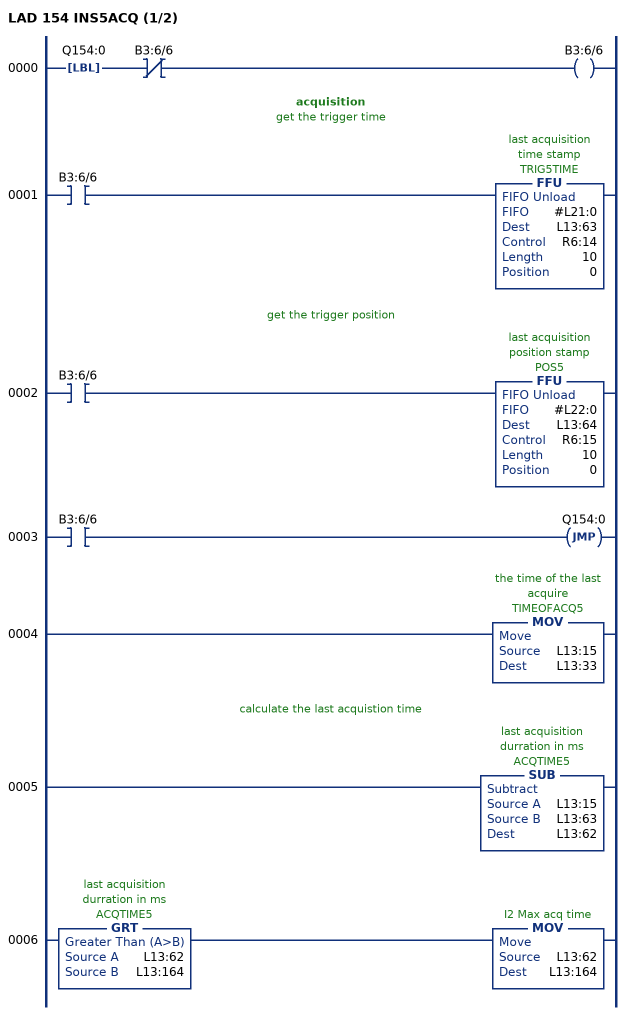
% Rung: 0 %
SOR LBL Q154:0 XIO B3:6/6 OTE B3:6/6 EOR
% Rung: 1 %
% TITLE: acquisition %
% get the trigger time %
SOR XIC B3:6/6 FFU #L21:0 L13:63 R6:14 10 0 EOR
%   L13:63  TRIG5TIME  "last acquisition time stamp" %
% Rung: 2 %
% get the trigger position %
SOR XIC B3:6/6 FFU #L22:0 L13:64 R6:15 10 0 EOR
%   L13:64  POS5  "last acquisition position stamp" %
% Rung: 3 %
SOR XIC B3:6/6 JMP Q154:0 EOR
% Rung: 4 %
SOR MOV L13:15 L13:33 EOR
%   L13:15  THE_TIME %
%   L13:33  TIMEOFACQ5  "the time of the last acquire" %
% Rung: 5 %
% calculate the last acquistion time %
SOR SUB L13:15 L13:63 L13:62 EOR
%   L13:15  THE_TIME %
%   L13:63  TRIG5TIME  "last acquisition time stamp" %
%   L13:62  ACQTIME5  "last acquisition durration in ms" %
% Rung: 6 %
SOR GRT L13:62 L13:164 MOV L13:62 L13:164 EOR
%   L13:62  ACQTIME5  "last acquisition durration in ms" %
%   L13:164  "I2 Max acq time" %

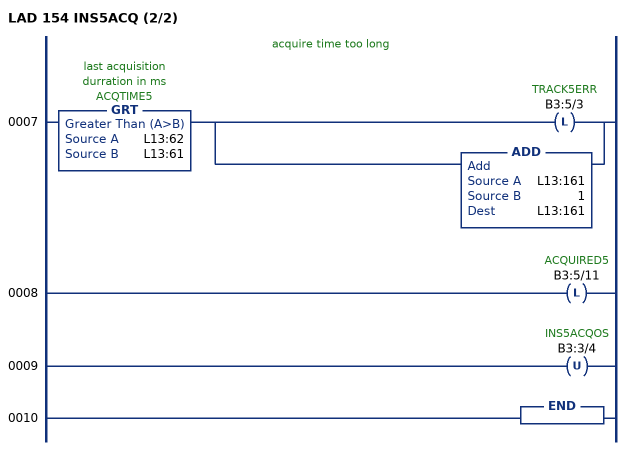
% Rung: 7 %
% acquire time too long %
SOR GRT L13:62 L13:61 BST OTL B3:5/3 NXB ADD L13:161 1 L13:161 BND EOR
%   L13:62  ACQTIME5  "last acquisition durration in ms" %
%   L13:61  "max acquisition time in ms" %
%   B3:5/3  TRACK5ERR %
% Rung: 8 %
SOR OTL B3:5/11 EOR
%   B3:5/11  ACQUIRED5 %
% Rung: 9 %
SOR OTU B3:3/4 EOR
%   B3:3/4  INS5ACQOS %
% Rung: 10 %
SOR END EOR

LADDER 155 "INS5TRIG"
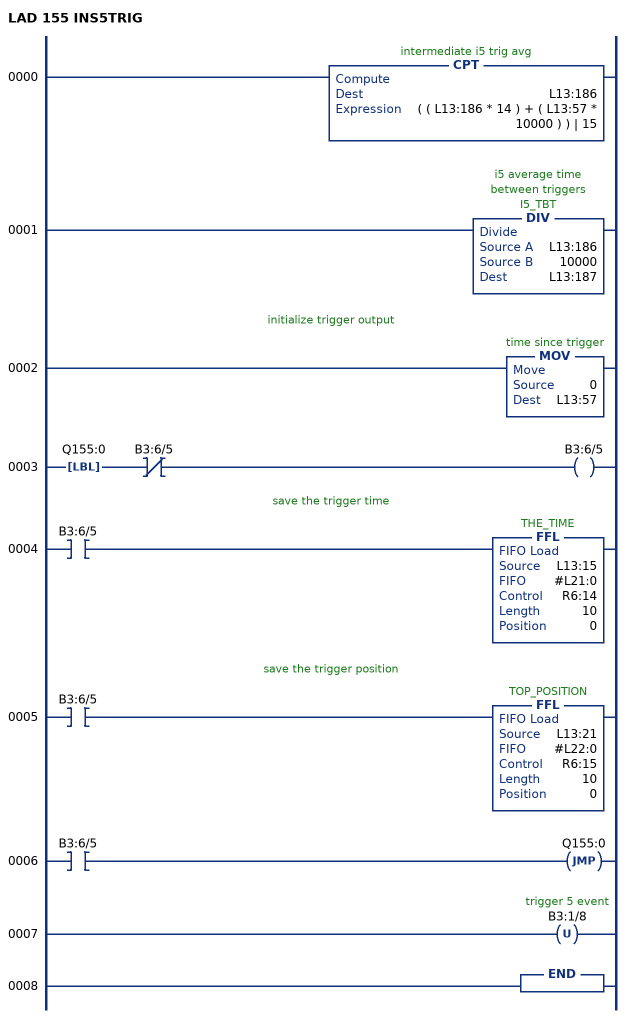
% Rung: 0 %
SOR CPT L13:186 " ( ( L13:186 * 14 ) + ( L13:57 * 10000 ) ) | 15 " EOR
%   L13:186  "intermediate i5 trig avg" %
%   L13:57  "time since trigger" %
% Rung: 1 %
SOR DIV L13:186 10000 L13:187 EOR
%   L13:186  "intermediate i5 trig avg" %
%   L13:187  I5_TBT  "i5 average time between triggers" %
% Rung: 2 %
% initialize trigger output %
SOR MOV 0 L13:57 EOR
%   L13:57  "time since trigger" %
% Rung: 3 %
SOR LBL Q155:0 XIO B3:6/5 OTE B3:6/5 EOR
% Rung: 4 %
% save the trigger time %
SOR XIC B3:6/5 FFL L13:15 #L21:0 R6:14 10 0 EOR
%   L13:15  THE_TIME %
% Rung: 5 %
% save the trigger position %
SOR XIC B3:6/5 FFL L13:21 #L22:0 R6:15 10 0 EOR
%   L13:21  TOP_POSITION %
% Rung: 6 %
SOR XIC B3:6/5 JMP Q155:0 EOR
% Rung: 7 %
SOR OTU B3:1/8 EOR
%   B3:1/8  "trigger 5 event" %
% Rung: 8 %
SOR END EOR

LADDER 159 "INS6RESULT"
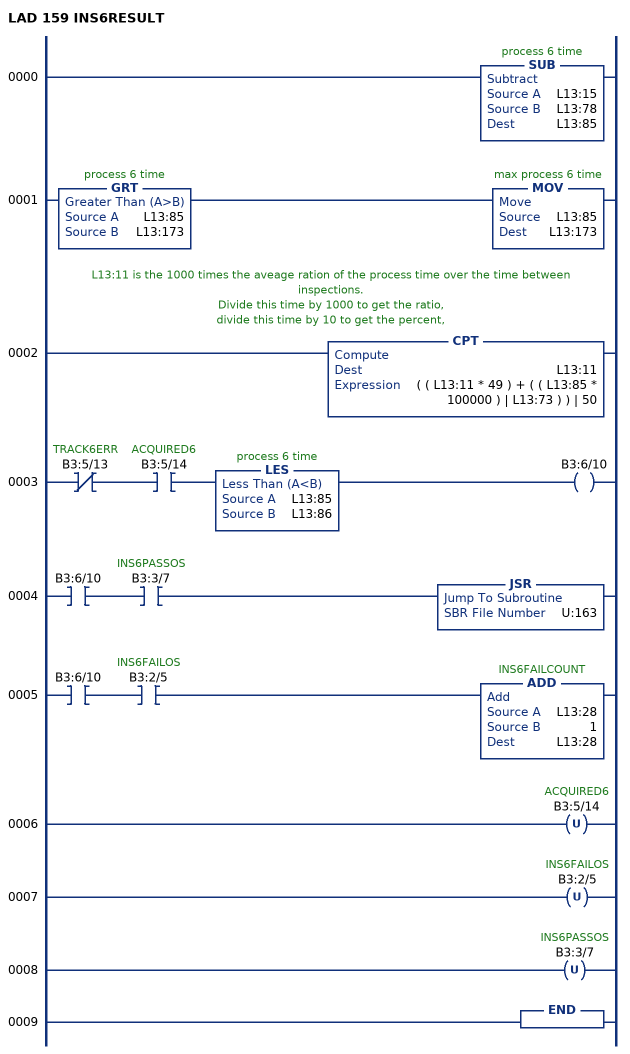
% Rung: 0 %
SOR SUB L13:15 L13:78 L13:85 EOR
%   L13:15  THE_TIME %
%   L13:78  TIMEOFACQ6  "the time of the last acquire" %
%   L13:85  "process 6 time" %
% Rung: 1 %
SOR GRT L13:85 L13:173 MOV L13:85 L13:173 EOR
%   L13:85  "process 6 time" %
%   L13:173  "max process 6 time" %
% Rung: 2 %
% L13:11 is the 1000 times the aveage ration of the process time over the time between inspections.
% Divide this time by 1000 to get the ratio,
% divide this time by 10 to get the percent, %
SOR CPT L13:11 " ( ( L13:11 * 49 ) + ( ( L13:85 * 100000 ) | L13:73 ) ) | 50 " EOR
%   L13:85  "process 6 time" %
%   L13:73  TBI  "the time between inspections in 0.000,01 seconds or 1/6000000 minutes." %
% Rung: 3 %
SOR XIO B3:5/13 XIC B3:5/14 LES L13:85 L13:86 OTE B3:6/10 EOR
%   B3:5/13  TRACK6ERR %
%   B3:5/14  ACQUIRED6 %
%   L13:85  "process 6 time" %
% Rung: 4 %
SOR XIC B3:6/10 XIC B3:3/7 JSR U:163 EOR
%   B3:3/7  INS6PASSOS %
% Rung: 5 %
SOR XIC B3:6/10 XIC B3:2/5 ADD L13:28 1 L13:28 EOR
%   B3:2/5  INS6FAILOS %
%   L13:28  INS6FAILCOUNT %
% Rung: 6 %
SOR OTU B3:5/14 EOR
%   B3:5/14  ACQUIRED6 %
% Rung: 7 %
SOR OTU B3:2/5 EOR
%   B3:2/5  INS6FAILOS %
% Rung: 8 %
SOR OTU B3:3/7 EOR
%   B3:3/7  INS6PASSOS %
% Rung: 9 %
SOR END EOR

LADDER 160 "FIXERR6"
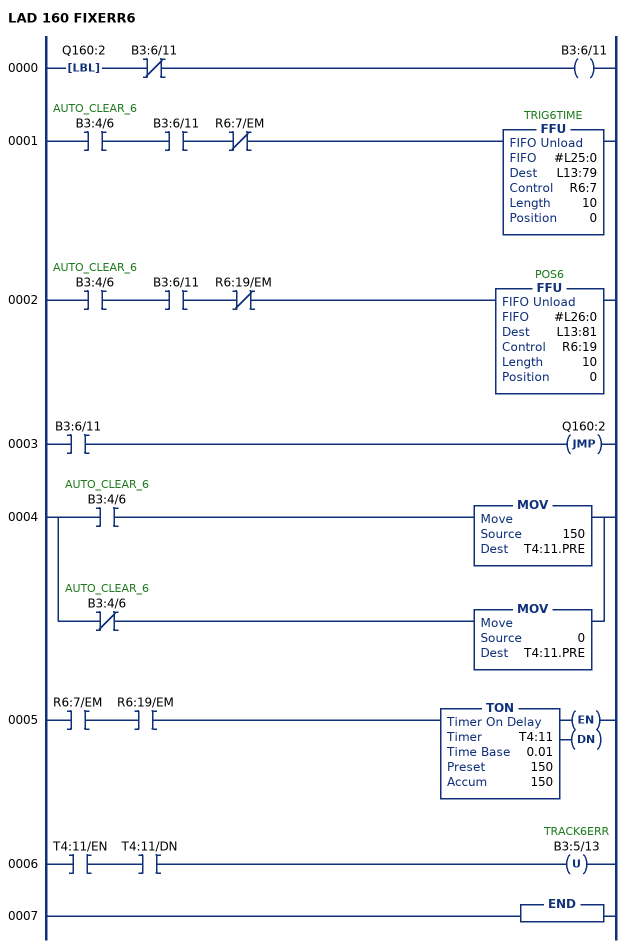
% Rung: 0 %
SOR LBL Q160:2 XIO B3:6/11 OTE B3:6/11 EOR
% Rung: 1 %
SOR XIC B3:4/6 XIC B3:6/11 XIO R6:7/EM FFU #L25:0 L13:79 R6:7 10 0 EOR
%   B3:4/6  AUTO_CLEAR_6 %
%   L13:79  TRIG6TIME %
% Rung: 2 %
SOR XIC B3:4/6 XIC B3:6/11 XIO R6:19/EM FFU #L26:0 L13:81 R6:19 10 0 EOR
%   B3:4/6  AUTO_CLEAR_6 %
%   L13:81  POS6 %
% Rung: 3 %
SOR XIC B3:6/11 JMP Q160:2 EOR
% Rung: 4 %
SOR BST XIC B3:4/6 MOV 150 T4:11.PRE NXB XIO B3:4/6 MOV 0 T4:11.PRE BND EOR
%   B3:4/6  AUTO_CLEAR_6 %
% Rung: 5 %
SOR XIC R6:7/EM XIC R6:19/EM TON T4:11 0.01 150 150 EOR
% Rung: 6 %
SOR XIC T4:11/EN XIC T4:11/DN OTU B3:5/13 EOR
%   B3:5/13  TRACK6ERR %
% Rung: 7 %
SOR END EOR

LADDER 162 "INS6"
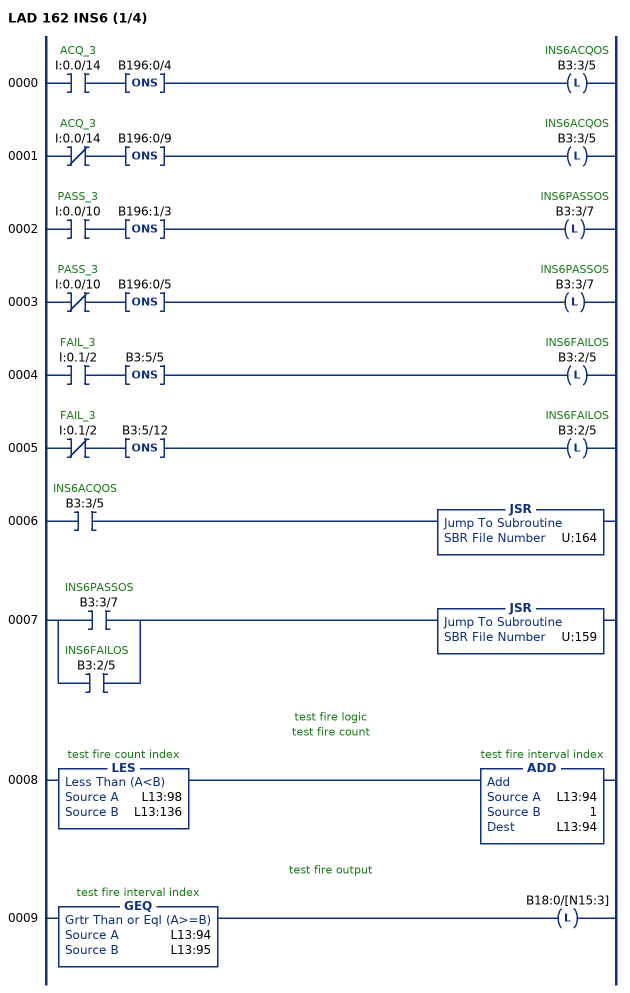
% Rung: 0 %
SOR XIC I:0.0/14 ONS B196:0/4 OTL B3:3/5 EOR
%   I:0.0/14  ACQ_3 %
%   B3:3/5  INS6ACQOS %
% Rung: 1 %
SOR XIO I:0.0/14 ONS B196:0/9 OTL B3:3/5 EOR
%   I:0.0/14  ACQ_3 %
%   B3:3/5  INS6ACQOS %
% Rung: 2 %
SOR XIC I:0.0/10 ONS B196:1/3 OTL B3:3/7 EOR
%   I:0.0/10  PASS_3 %
%   B3:3/7  INS6PASSOS %
% Rung: 3 %
SOR XIO I:0.0/10 ONS B196:0/5 OTL B3:3/7 EOR
%   I:0.0/10  PASS_3 %
%   B3:3/7  INS6PASSOS %
% Rung: 4 %
SOR XIC I:0.1/2 ONS B3:5/5 OTL B3:2/5 EOR
%   I:0.1/2  FAIL_3 %
%   B3:2/5  INS6FAILOS %
% Rung: 5 %
SOR XIO I:0.1/2 ONS B3:5/12 OTL B3:2/5 EOR
%   I:0.1/2  FAIL_3 %
%   B3:2/5  INS6FAILOS %
% Rung: 6 %
SOR XIC B3:3/5 JSR U:164 EOR
%   B3:3/5  INS6ACQOS %
% Rung: 7 %
SOR BST XIC B3:3/7 NXB XIC B3:2/5 BND JSR U:159 EOR
%   B3:3/7  INS6PASSOS %
%   B3:2/5  INS6FAILOS %
% Rung: 8 %
% test fire logic
% 
% test fire count %
SOR LES L13:98 L13:136 ADD L13:94 1 L13:94 EOR
%   L13:98  "test fire count index" %
%   L13:136  "test fire count" %
%   L13:94  "test fire interval index" %
% Rung: 9 %
% test fire output %
SOR GEQ L13:94 L13:95 OTL B18:0/[N15:3] EOR
%   L13:94  "test fire interval index" %
%   L13:95  "test fire interval" %
%   N15:3  INS_6_TRIG_LOC %

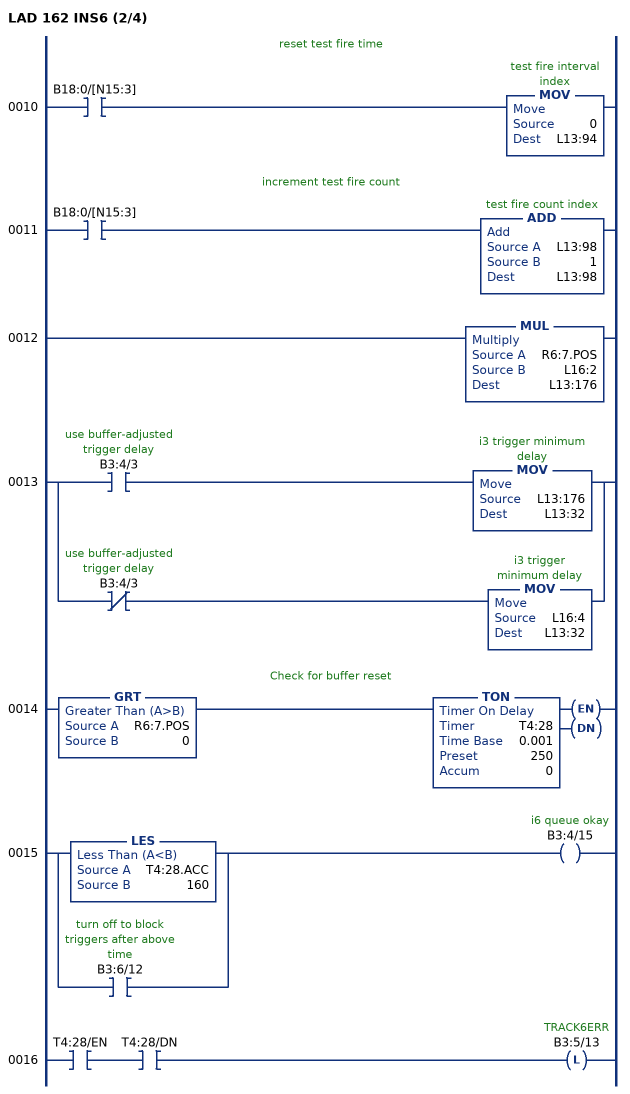
% Rung: 10 %
% reset test fire time %
SOR XIC B18:0/[N15:3] MOV 0 L13:94 EOR
%   N15:3  INS_6_TRIG_LOC %
%   L13:94  "test fire interval index" %
% Rung: 11 %
% increment test fire count %
SOR XIC B18:0/[N15:3] ADD L13:98 1 L13:98 EOR
%   N15:3  INS_6_TRIG_LOC %
%   L13:98  "test fire count index" %
% Rung: 12 %
SOR MUL R6:7.POS L16:2 L13:176 EOR
%   L16:2  TRIG_DELAY_Q_MULTI %
% Rung: 13 %
SOR BST XIC B3:4/3 MOV L13:176 L13:32 NXB XIO B3:4/3 MOV L16:4 L13:32 BND EOR
%   B3:4/3  "use buffer-adjusted trigger delay" %
%   L13:32  "i3 trigger minimum delay" %
%   L16:4  TRIG_DELAY_FLAT_RATE %
% Rung: 14 %
% Check for buffer reset %
SOR GRT R6:7.POS 0 TON T4:28 0.001 250 0 EOR
% Rung: 15 %
SOR BST LES T4:28.ACC 160 NXB XIC B3:6/12 BND OTE B3:4/15 EOR
%   B3:6/12  "turn off to block triggers after above time" %
%   B3:4/15  "i6 queue okay" %
% Rung: 16 %
SOR XIC T4:28/EN XIC T4:28/DN OTL B3:5/13 EOR
%   B3:5/13  TRACK6ERR %

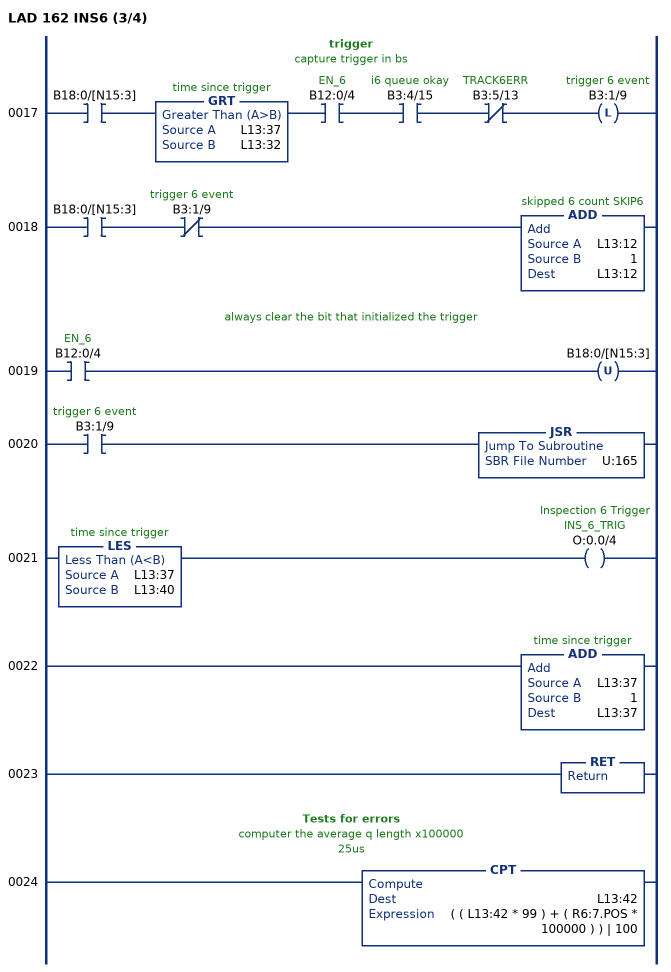
% Rung: 17 %
% TITLE: trigger %
% capture trigger in bs %
SOR XIC B18:0/[N15:3] GRT L13:37 L13:32 XIC B12:0/4 XIC B3:4/15 XIO B3:5/13 OTL B3:1/9 EOR
%   N15:3  INS_6_TRIG_LOC %
%   L13:37  "time since trigger" %
%   L13:32  "i3 trigger minimum delay" %
%   B12:0/4  EN_6 %
%   B3:4/15  "i6 queue okay" %
%   B3:5/13  TRACK6ERR %
%   B3:1/9  "trigger 6 event" %
% Rung: 18 %
SOR XIC B18:0/[N15:3] XIO B3:1/9 ADD L13:12 1 L13:12 EOR
%   N15:3  INS_6_TRIG_LOC %
%   B3:1/9  "trigger 6 event" %
%   L13:12  SKIP6  "skipped 6 count" %
% Rung: 19 %
% always clear the bit that initialized the trigger %
SOR XIC B12:0/4 OTU B18:0/[N15:3] EOR
%   B12:0/4  EN_6 %
%   N15:3  INS_6_TRIG_LOC %
% Rung: 20 %
SOR XIC B3:1/9 JSR U:165 EOR
%   B3:1/9  "trigger 6 event" %
% Rung: 21 %
SOR LES L13:37 L13:40 OTE O:0.0/4 EOR
%   L13:37  "time since trigger" %
%   L13:40  "last part time" %
%   O:0.0/4  INS_6_TRIG  "Inspection 6 Trigger" %
% Rung: 22 %
SOR ADD L13:37 1 L13:37 EOR
%   L13:37  "time since trigger" %
% Rung: 23 %
SOR RET EOR
% Rung: 24 %
% TITLE: Tests for errors %
% computer the average q length x100000
% 25us %
SOR CPT L13:42 " ( ( L13:42 * 99 ) + ( R6:7.POS * 100000 ) ) | 100 " EOR

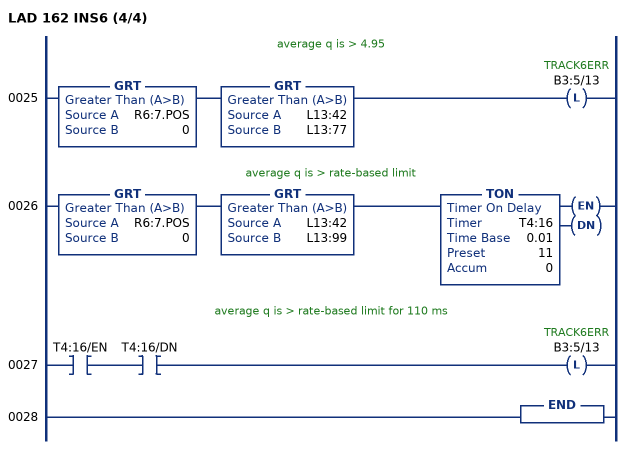
% Rung: 25 %
% average q is > 4.95 %
SOR GRT R6:7.POS 0 GRT L13:42 L13:77 OTL B3:5/13 EOR
%   B3:5/13  TRACK6ERR %
% Rung: 26 %
% average q is > rate-based limit %
SOR GRT R6:7.POS 0 GRT L13:42 L13:99 TON T4:16 0.01 11 0 EOR
%   L13:99  "i6 timed queue limit" %
% Rung: 27 %
% average q is > rate-based limit for 110 ms %
SOR XIC T4:16/EN XIC T4:16/DN OTL B3:5/13 EOR
%   B3:5/13  TRACK6ERR %
% Rung: 28 %
SOR END EOR

LADDER 163 "INS6PASS"
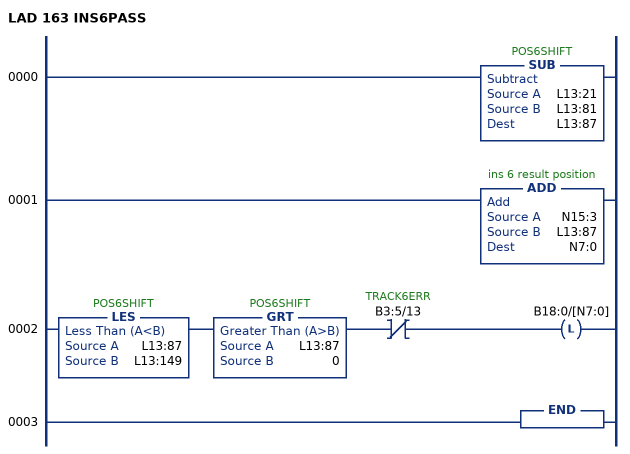
% Rung: 0 %
SOR SUB L13:21 L13:81 L13:87 EOR
%   L13:21  TOP_POSITION %
%   L13:81  POS6 %
%   L13:87  POS6SHIFT %
% Rung: 1 %
SOR ADD N15:3 L13:87 N7:0 EOR
%   N15:3  INS_6_TRIG_LOC %
%   L13:87  POS6SHIFT %
%   N7:0  "ins 6 result position" %
% Rung: 2 %
SOR LES L13:87 L13:149 GRT L13:87 0 XIO B3:5/13 OTL B18:0/[N7:0] EOR
%   L13:87  POS6SHIFT %
%   B3:5/13  TRACK6ERR %
%   N7:0  "ins 6 result position" %
% Rung: 3 %
SOR END EOR

LADDER 164 "INS6ACQ"
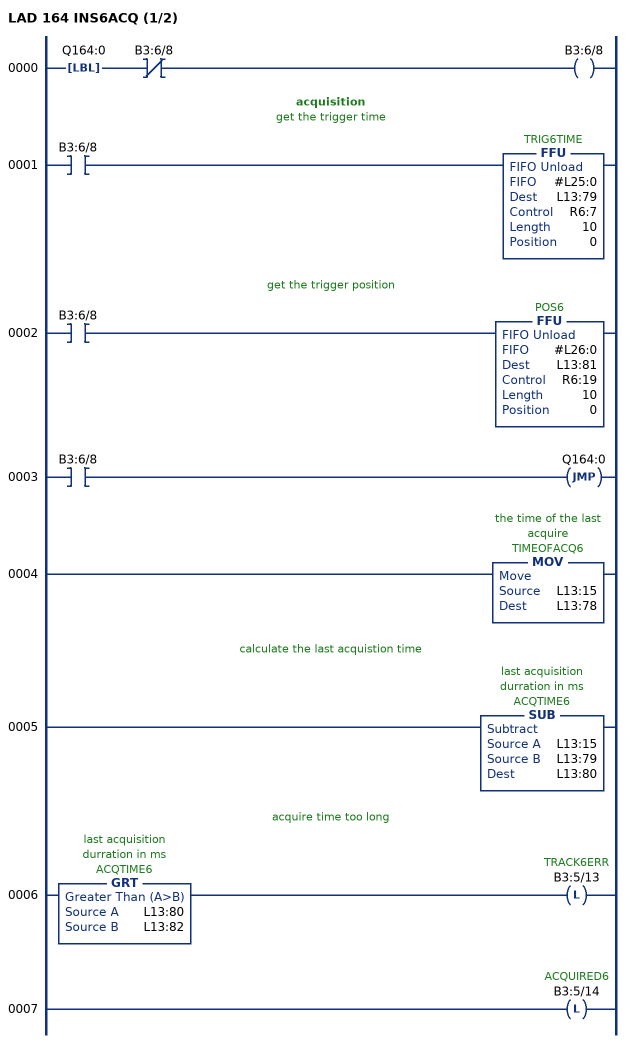
% Rung: 0 %
SOR LBL Q164:0 XIO B3:6/8 OTE B3:6/8 EOR
% Rung: 1 %
% TITLE: acquisition %
% get the trigger time %
SOR XIC B3:6/8 FFU #L25:0 L13:79 R6:7 10 0 EOR
%   L13:79  TRIG6TIME %
% Rung: 2 %
% get the trigger position %
SOR XIC B3:6/8 FFU #L26:0 L13:81 R6:19 10 0 EOR
%   L13:81  POS6 %
% Rung: 3 %
SOR XIC B3:6/8 JMP Q164:0 EOR
% Rung: 4 %
SOR MOV L13:15 L13:78 EOR
%   L13:15  THE_TIME %
%   L13:78  TIMEOFACQ6  "the time of the last acquire" %
% Rung: 5 %
% calculate the last acquistion time %
SOR SUB L13:15 L13:79 L13:80 EOR
%   L13:15  THE_TIME %
%   L13:79  TRIG6TIME %
%   L13:80  ACQTIME6  "last acquisition durration in ms" %
% Rung: 6 %
% acquire time too long %
SOR GRT L13:80 L13:82 OTL B3:5/13 EOR
%   L13:80  ACQTIME6  "last acquisition durration in ms" %
%   B3:5/13  TRACK6ERR %
% Rung: 7 %
SOR OTL B3:5/14 EOR
%   B3:5/14  ACQUIRED6 %

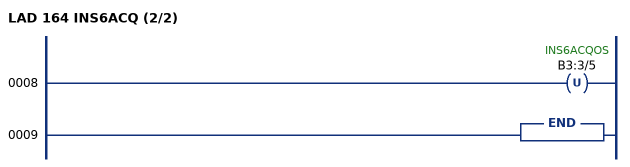
% Rung: 8 %
SOR OTU B3:3/5 EOR
%   B3:3/5  INS6ACQOS %
% Rung: 9 %
SOR END EOR

LADDER 165 "INS6TRIG"
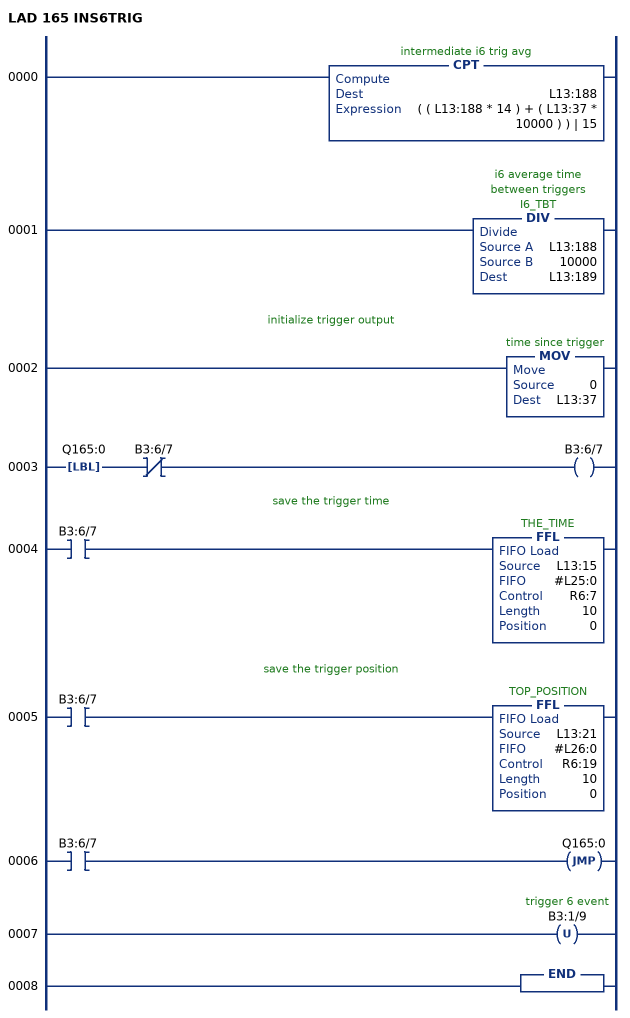
% Rung: 0 %
SOR CPT L13:188 " ( ( L13:188 * 14 ) + ( L13:37 * 10000 ) ) | 15 " EOR
%   L13:188  "intermediate i6 trig avg" %
%   L13:37  "time since trigger" %
% Rung: 1 %
SOR DIV L13:188 10000 L13:189 EOR
%   L13:188  "intermediate i6 trig avg" %
%   L13:189  I6_TBT  "i6 average time between triggers" %
% Rung: 2 %
% initialize trigger output %
SOR MOV 0 L13:37 EOR
%   L13:37  "time since trigger" %
% Rung: 3 %
SOR LBL Q165:0 XIO B3:6/7 OTE B3:6/7 EOR
% Rung: 4 %
% save the trigger time %
SOR XIC B3:6/7 FFL L13:15 #L25:0 R6:7 10 0 EOR
%   L13:15  THE_TIME %
% Rung: 5 %
% save the trigger position %
SOR XIC B3:6/7 FFL L13:21 #L26:0 R6:19 10 0 EOR
%   L13:21  TOP_POSITION %
% Rung: 6 %
SOR XIC B3:6/7 JMP Q165:0 EOR
% Rung: 7 %
SOR OTU B3:1/9 EOR
%   B3:1/9  "trigger 6 event" %
% Rung: 8 %
SOR END EOR

LADDER 170 "PASS BLOW"
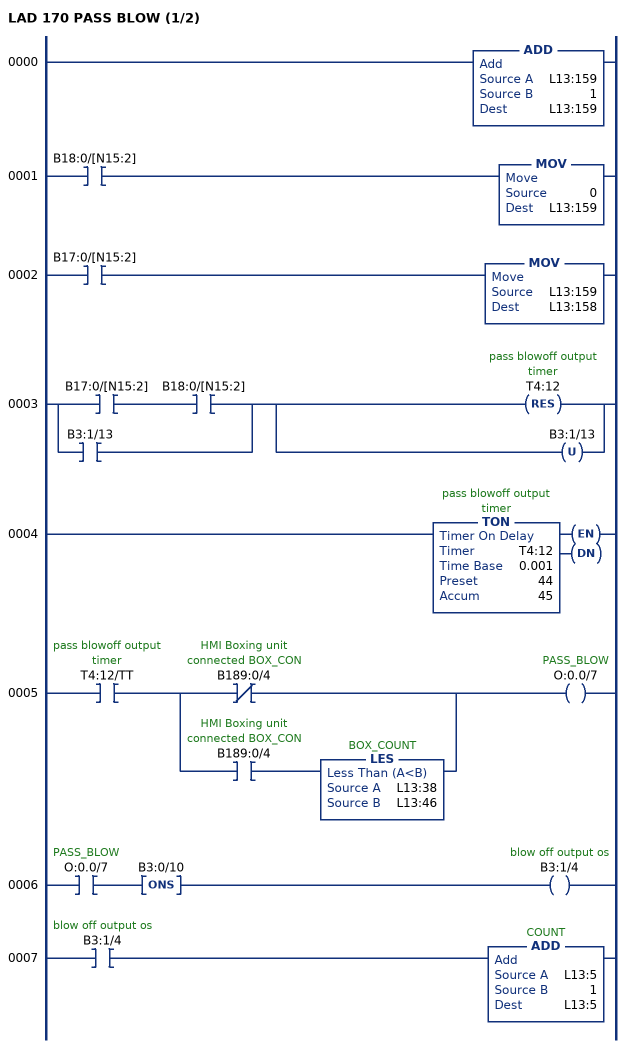
% Rung: 0 %
SOR ADD L13:159 1 L13:159 EOR
% Rung: 1 %
SOR XIC B18:0/[N15:2] MOV 0 L13:159 EOR
%   N15:2  BLOW_PT %
% Rung: 2 %
SOR XIC B17:0/[N15:2] MOV L13:159 L13:158 EOR
%   N15:2  BLOW_PT %
% Rung: 3 %
SOR BST XIC B17:0/[N15:2] XIC B18:0/[N15:2] NXB XIC B3:1/13 BND BST RES T4:12 NXB OTU B3:1/13 BND EOR
%   N15:2  BLOW_PT %
%   T4:12  "pass blowoff output timer" %
% Rung: 4 %
SOR TON T4:12 0.001 44 45 EOR
%   T4:12  "pass blowoff output timer" %
% Rung: 5 %
SOR XIC T4:12/TT BST XIO B189:0/4 NXB XIC B189:0/4 LES L13:38 L13:46 BND OTE O:0.0/7 EOR
%   T4:12  "pass blowoff output timer" %
%   B189:0/4  BOX_CON  "HMI Boxing unit connected" %
%   L13:38  BOX_COUNT %
%   L13:46  BOX_LIMIT  "box count setpoint" %
%   O:0.0/7  PASS_BLOW %
% Rung: 6 %
SOR XIC O:0.0/7 ONS B3:0/10 OTE B3:1/4 EOR
%   O:0.0/7  PASS_BLOW %
%   B3:1/4  "blow off output os" %
% Rung: 7 %
SOR XIC B3:1/4 ADD L13:5 1 L13:5 EOR
%   B3:1/4  "blow off output os" %
%   L13:5  COUNT %

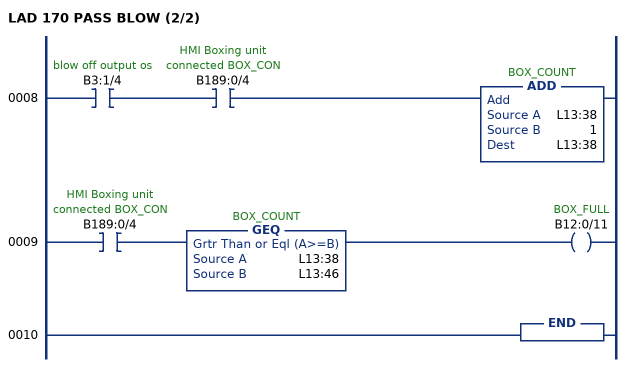
% Rung: 8 %
SOR XIC B3:1/4 XIC B189:0/4 ADD L13:38 1 L13:38 EOR
%   B3:1/4  "blow off output os" %
%   B189:0/4  BOX_CON  "HMI Boxing unit connected" %
%   L13:38  BOX_COUNT %
% Rung: 9 %
SOR XIC B189:0/4 GEQ L13:38 L13:46 OTE B12:0/11 EOR
%   B189:0/4  BOX_CON  "HMI Boxing unit connected" %
%   L13:38  BOX_COUNT %
%   L13:46  BOX_LIMIT  "box count setpoint" %
%   B12:0/11  BOX_FULL %
% Rung: 10 %
SOR END EOR

LADDER 180 "RATE"
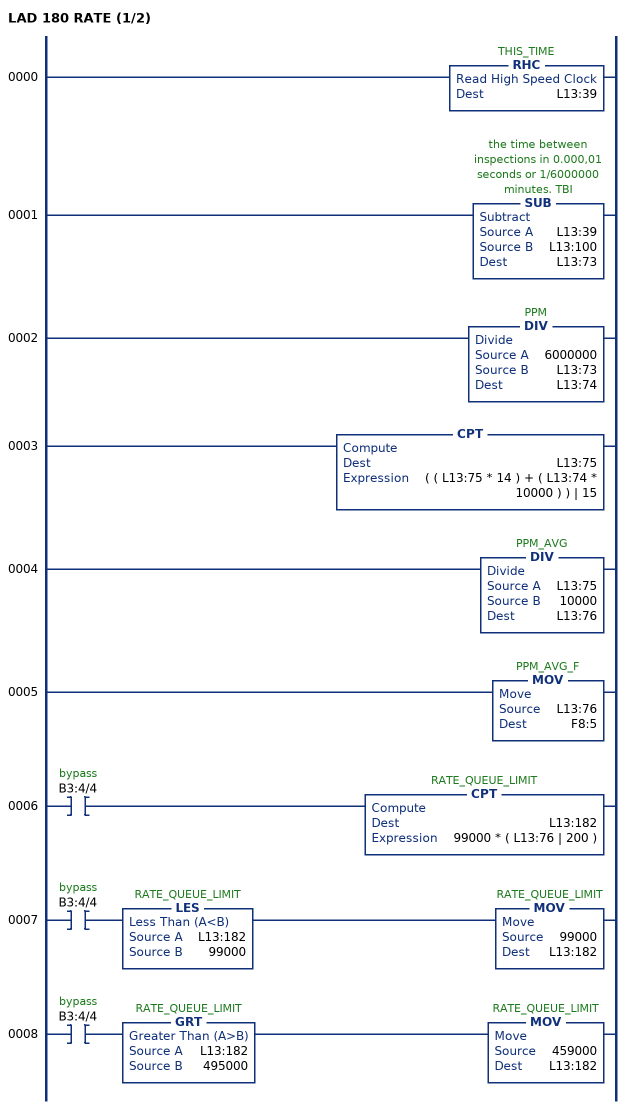
% Rung: 0 %
SOR RHC L13:39 EOR
%   L13:39  THIS_TIME %
% Rung: 1 %
SOR SUB L13:39 L13:100 L13:73 EOR
%   L13:39  THIS_TIME %
%   L13:100  LAST_PART_TIME  "the time clock reading when the previous part was triggered" %
%   L13:73  TBI  "the time between inspections in 0.000,01 seconds or 1/6000000 minutes." %
% Rung: 2 %
SOR DIV 6000000 L13:73 L13:74 EOR
%   L13:73  TBI  "the time between inspections in 0.000,01 seconds or 1/6000000 minutes." %
%   L13:74  PPM %
% Rung: 3 %
SOR CPT L13:75 " ( ( L13:75 * 14 ) + ( L13:74 * 10000 ) ) | 15 " EOR
%   L13:74  PPM %
% Rung: 4 %
SOR DIV L13:75 10000 L13:76 EOR
%   L13:76  PPM_AVG %
% Rung: 5 %
SOR MOV L13:76 F8:5 EOR
%   L13:76  PPM_AVG %
%   F8:5  PPM_AVG_F %
% Rung: 6 %
SOR XIC B3:4/4 CPT L13:182 " 99000 * ( L13:76 | 200 ) " EOR
%   B3:4/4  "bypass" %
%   L13:182  RATE_QUEUE_LIMIT %
%   L13:76  PPM_AVG %
% Rung: 7 %
SOR XIC B3:4/4 LES L13:182 99000 MOV 99000 L13:182 EOR
%   B3:4/4  "bypass" %
%   L13:182  RATE_QUEUE_LIMIT %
% Rung: 8 %
SOR XIC B3:4/4 GRT L13:182 495000 MOV 459000 L13:182 EOR
%   B3:4/4  "bypass" %
%   L13:182  RATE_QUEUE_LIMIT %

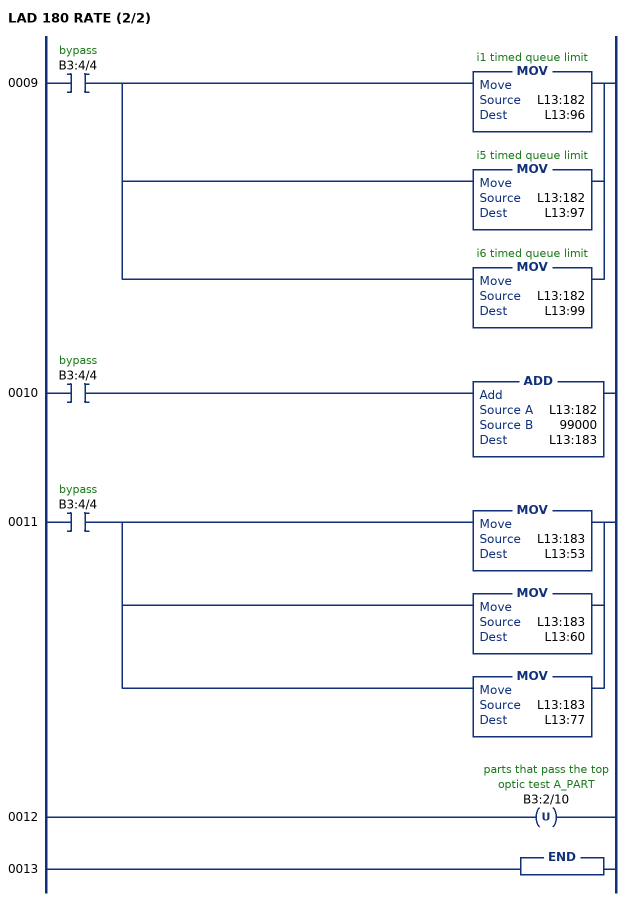
% Rung: 9 %
SOR XIC B3:4/4 BST MOV L13:182 L13:96 NXB MOV L13:182 L13:97 NXB MOV L13:182 L13:99 BND EOR
%   B3:4/4  "bypass" %
%   L13:182  RATE_QUEUE_LIMIT %
%   L13:96  "i1 timed queue limit" %
%   L13:97  "i5 timed queue limit" %
%   L13:99  "i6 timed queue limit" %
% Rung: 10 %
SOR XIC B3:4/4 ADD L13:182 99000 L13:183 EOR
%   B3:4/4  "bypass" %
%   L13:182  RATE_QUEUE_LIMIT %
% Rung: 11 %
SOR XIC B3:4/4 BST MOV L13:183 L13:53 NXB MOV L13:183 L13:60 NXB MOV L13:183 L13:77 BND EOR
%   B3:4/4  "bypass" %
% Rung: 12 %
SOR OTU B3:2/10 EOR
%   B3:2/10  A_PART  "parts that pass the top optic test" %
% Rung: 13 %
SOR END EOR

LADDER 200 "TESTOPTIC"
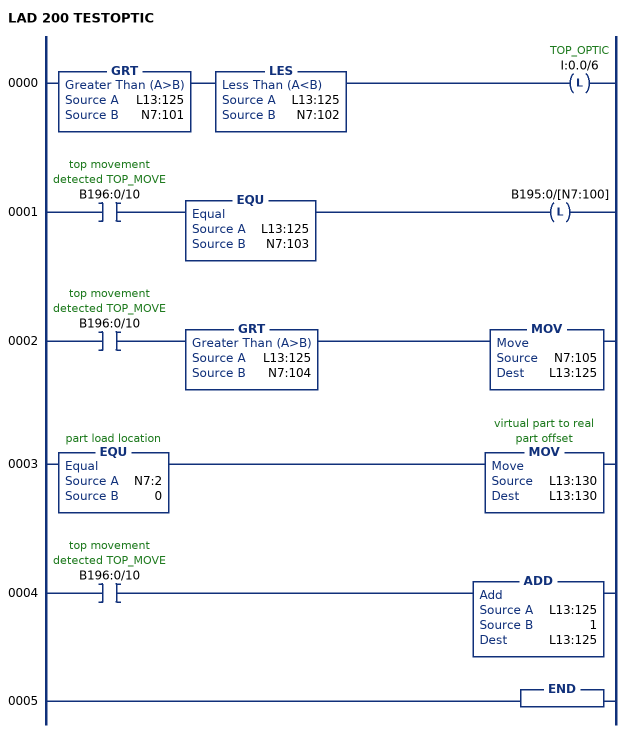
% Rung: 0 %
SOR GRT L13:125 N7:101 LES L13:125 N7:102 OTL I:0.0/6 EOR
%   I:0.0/6  TOP_OPTIC %
% Rung: 1 %
SOR XIC B196:0/10 EQU L13:125 N7:103 OTL B195:0/[N7:100] EOR
%   B196:0/10  TOP_MOVE  "top movement detected" %
% Rung: 2 %
SOR XIC B196:0/10 GRT L13:125 N7:104 MOV N7:105 L13:125 EOR
%   B196:0/10  TOP_MOVE  "top movement detected" %
% Rung: 3 %
SOR EQU N7:2 0 MOV L13:130 L13:130 EOR
%   N7:2  "part load location" %
%   L13:130  "virtual part to real part offset" %
% Rung: 4 %
SOR XIC B196:0/10 ADD L13:125 1 L13:125 EOR
%   B196:0/10  TOP_MOVE  "top movement detected" %
% Rung: 5 %
SOR END EOR

LADDER 201 "UNUSED"
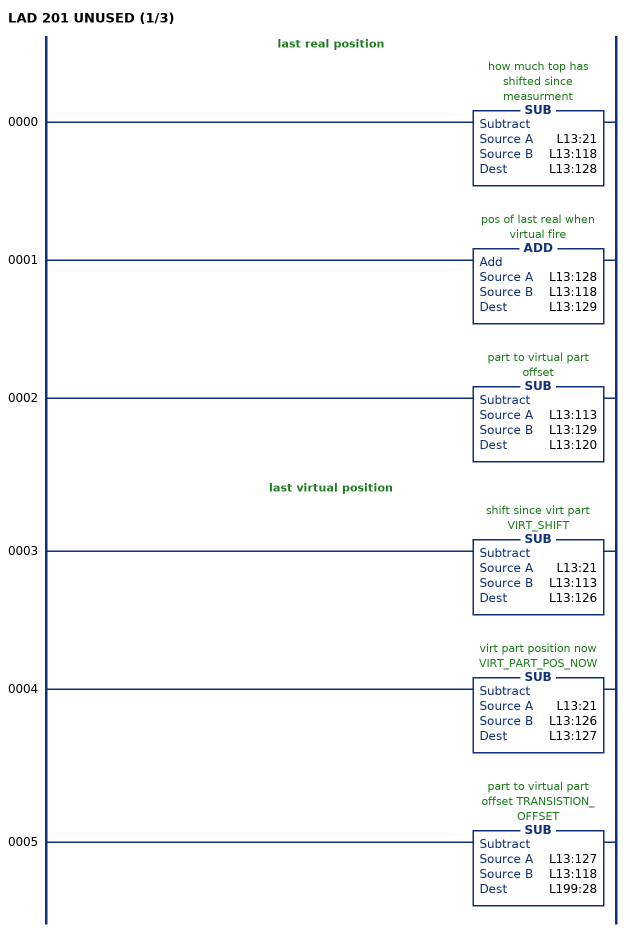
% Rung: 0 %
% TITLE: last real position %
SOR SUB L13:21 L13:118 L13:128 EOR
%   L13:21  TOP_POSITION %
%   L13:118  REAL_PT_RAW_CL  "real part center line in raw position" %
%   L13:128  "how much top has shifted since measurment" %
% Rung: 1 %
SOR ADD L13:128 L13:118 L13:129 EOR
%   L13:128  "how much top has shifted since measurment" %
%   L13:118  REAL_PT_RAW_CL  "real part center line in raw position" %
%   L13:129  "pos of last real when virtual fire" %
% Rung: 2 %
SOR SUB L13:113 L13:129 L13:120 EOR
%   L13:113  VERTUAL_PT_RAW_CL  "virtual part center line transfer from the bottom in raw position" %
%   L13:129  "pos of last real when virtual fire" %
%   L13:120  "part to virtual part offset" %
% Rung: 3 %
% TITLE: last virtual position %
SOR SUB L13:21 L13:113 L13:126 EOR
%   L13:21  TOP_POSITION %
%   L13:113  VERTUAL_PT_RAW_CL  "virtual part center line transfer from the bottom in raw position" %
%   L13:126  VIRT_SHIFT  "shift since virt part" %
% Rung: 4 %
SOR SUB L13:21 L13:126 L13:127 EOR
%   L13:21  TOP_POSITION %
%   L13:126  VIRT_SHIFT  "shift since virt part" %
%   L13:127  VIRT_PART_POS_NOW  "virt part position now" %
% Rung: 5 %
SOR SUB L13:127 L13:118 L199:28 EOR
%   L13:127  VIRT_PART_POS_NOW  "virt part position now" %
%   L13:118  REAL_PT_RAW_CL  "real part center line in raw position" %
%   L199:28  TRANSISTION_OFFSET  "part to virtual part offset" %

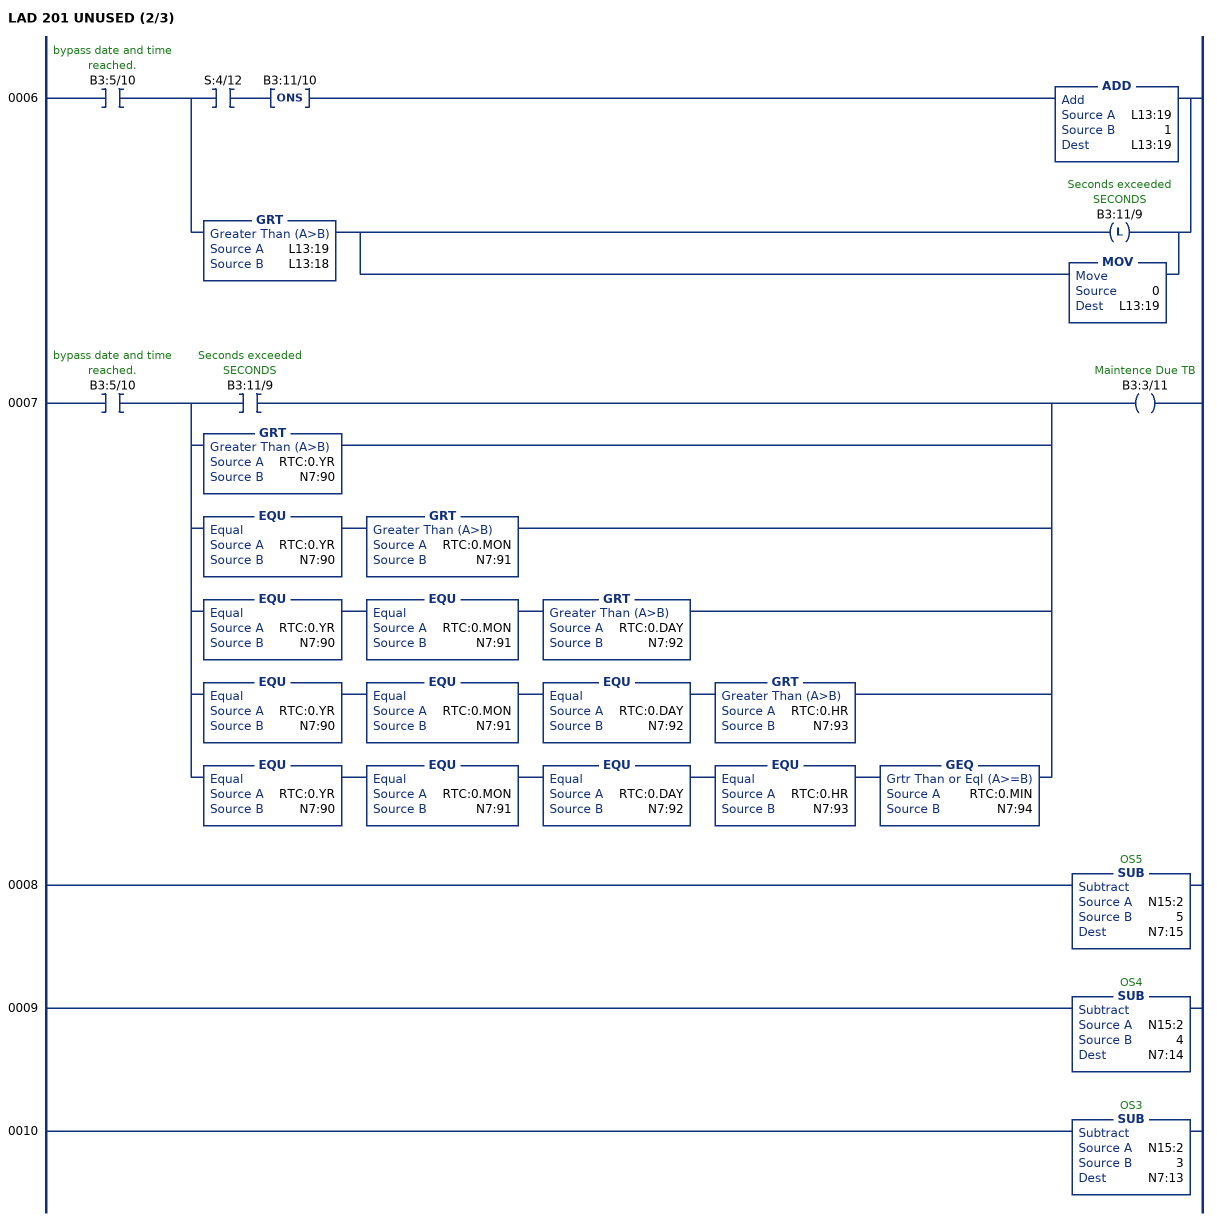
% Rung: 6 %
SOR XIC B3:5/10 BST XIC S:4/12 ONS B3:11/10 ADD L13:19 1 L13:19 NXB GRT L13:19 L13:18 BST OTL B3:11/9 NXB MOV 0 L13:19 BND BND EOR
%   B3:5/10  "bypass date and time reached." %
%   L13:18  MAX %
%   B3:11/9  SECONDS  "Seconds exceeded" %
% Rung: 7 %
SOR XIC B3:5/10 BST XIC B3:11/9 NXB GRT RTC:0.YR N7:90 NXB EQU RTC:0.YR N7:90 GRT RTC:0.MON N7:91 NXB EQU RTC:0.YR N7:90 EQU RTC:0.MON N7:91 GRT RTC:0.DAY N7:92 NXB EQU RTC:0.YR N7:90 EQU RTC:0.MON N7:91 EQU RTC:0.DAY N7:92 GRT RTC:0.HR N7:93 NXB EQU RTC:0.YR N7:90 EQU RTC:0.MON N7:91 EQU RTC:0.DAY N7:92 EQU RTC:0.HR N7:93 GEQ RTC:0.MIN N7:94 BND OTE B3:3/11 EOR
%   B3:5/10  "bypass date and time reached." %
%   B3:11/9  SECONDS  "Seconds exceeded" %
%   N7:90  RTC %
%   B3:3/11  TB  "Maintence Due" %
% Rung: 8 %
SOR SUB N15:2 5 N7:15 EOR
%   N15:2  BLOW_PT %
%   N7:15  OS5 %
% Rung: 9 %
SOR SUB N15:2 4 N7:14 EOR
%   N15:2  BLOW_PT %
%   N7:14  OS4 %
% Rung: 10 %
SOR SUB N15:2 3 N7:13 EOR
%   N15:2  BLOW_PT %
%   N7:13  OS3 %

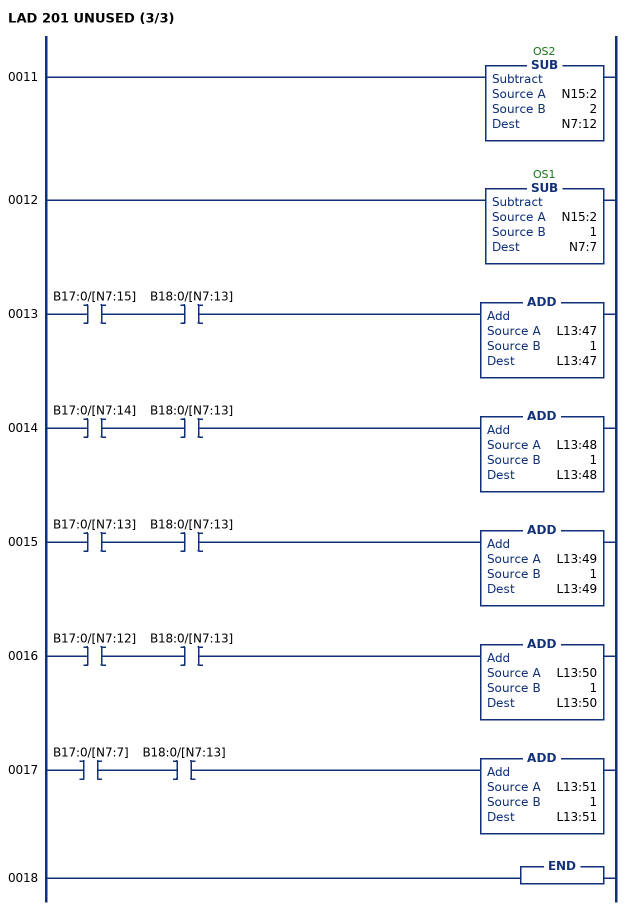
% Rung: 11 %
SOR SUB N15:2 2 N7:12 EOR
%   N15:2  BLOW_PT %
%   N7:12  OS2 %
% Rung: 12 %
SOR SUB N15:2 1 N7:7 EOR
%   N15:2  BLOW_PT %
%   N7:7  OS1 %
% Rung: 13 %
SOR XIC B17:0/[N7:15] XIC B18:0/[N7:13] ADD L13:47 1 L13:47 EOR
%   N7:15  OS5 %
%   N7:13  OS3 %
% Rung: 14 %
SOR XIC B17:0/[N7:14] XIC B18:0/[N7:13] ADD L13:48 1 L13:48 EOR
%   N7:14  OS4 %
%   N7:13  OS3 %
% Rung: 15 %
SOR XIC B17:0/[N7:13] XIC B18:0/[N7:13] ADD L13:49 1 L13:49 EOR
%   N7:13  OS3 %
% Rung: 16 %
SOR XIC B17:0/[N7:12] XIC B18:0/[N7:13] ADD L13:50 1 L13:50 EOR
%   N7:12  OS2 %
%   N7:13  OS3 %
% Rung: 17 %
SOR XIC B17:0/[N7:7] XIC B18:0/[N7:13] ADD L13:51 1 L13:51 EOR
%   N7:7  OS1 %
%   N7:13  OS3 %
% Rung: 18 %
SOR END EOR

LADDER 255 "BLANK"
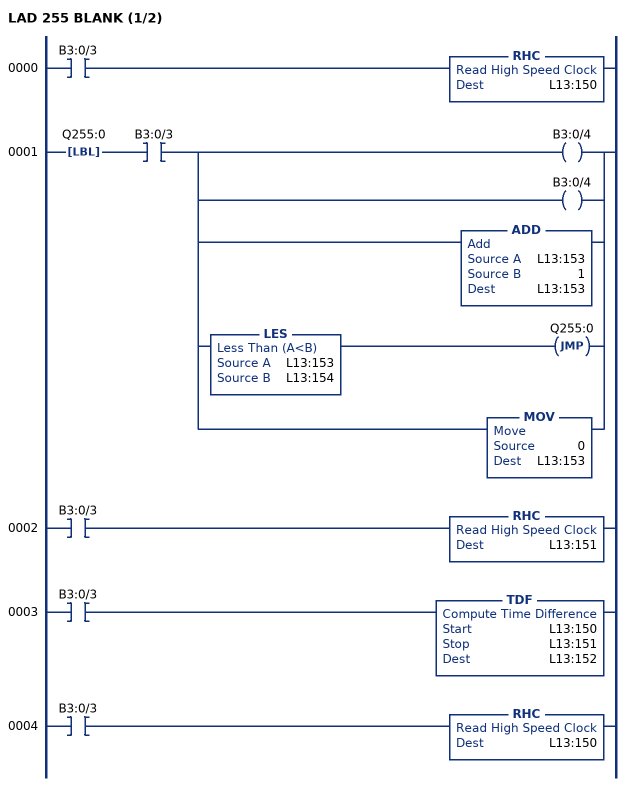
% Rung: 0 %
SOR XIC B3:0/3 RHC L13:150 EOR
% Rung: 1 %
SOR LBL Q255:0 XIC B3:0/3 BST OTE B3:0/4 NXB OTE B3:0/4 NXB ADD L13:153 1 L13:153 NXB LES L13:153 L13:154 JMP Q255:0 NXB MOV 0 L13:153 BND EOR
% Rung: 2 %
SOR XIC B3:0/3 RHC L13:151 EOR
% Rung: 3 %
SOR XIC B3:0/3 TDF L13:150 L13:151 L13:152 EOR
% Rung: 4 %
SOR XIC B3:0/3 RHC L13:150 EOR

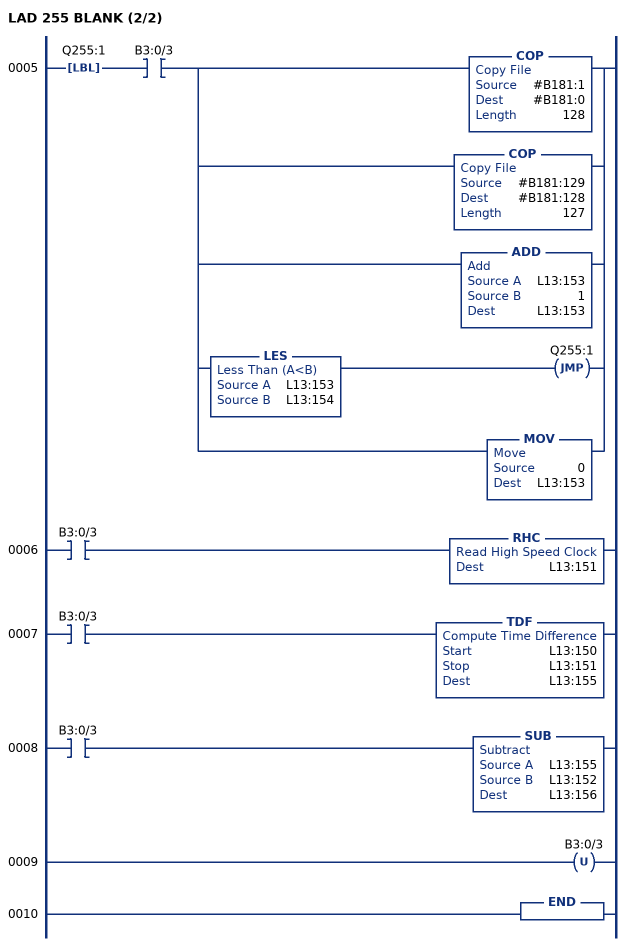
% Rung: 5 %
SOR LBL Q255:1 XIC B3:0/3 BST COP #B181:1 #B181:0 128 NXB COP #B181:129 #B181:128 127 NXB ADD L13:153 1 L13:153 NXB LES L13:153 L13:154 JMP Q255:1 NXB MOV 0 L13:153 BND EOR
% Rung: 6 %
SOR XIC B3:0/3 RHC L13:151 EOR
% Rung: 7 %
SOR XIC B3:0/3 TDF L13:150 L13:151 L13:155 EOR
% Rung: 8 %
SOR XIC B3:0/3 SUB L13:155 L13:152 L13:156 EOR
% Rung: 9 %
SOR OTU B3:0/3 EOR
% Rung: 10 %
SOR END EOR

OTHER DOCUMENTED ADDRESSES
  B3:10/14  "Dont use"
  BUL_COUNT_REACHED  
  HSC:0.0  "top"
  HSC:0.3/6  "Underflow interrupt"
  HSC:0.3/7  "Overflow interrupt"
  HSC:1.0  "bot"
  HSC:1.3/6  "Underflow interrupt"
  HSC:1.3/7  "Overflow interrupt"
  I:0.0/0  "Encoder Signal "A""
  I:0.0/1  "Encoder Signal "B""
  I:0.0/4  "Encoder Signal "A""
  I:0.0/5  "Encoder Signal "B""
  I:0.0/11  PASS_4
  I:0.0/15  ACQ_4
  I:0.1/3  FAIL_4
  I:0.2/3  "Packaging Conveyor full"
  I:0.2/4  "Packaging Conveyor Box in Position"
  I:0.4  "Spare Analog Input 1"
  I:0.5  "Spare Analog Input 2"
  I:0.6  "Spare Analog Input 3"
  I:2.0/1  REAR_ESTOP
  I:2.0/8  "front door signal"
  I:2.0/9  "rear door signal"
  I:2.0/10  "Maintenance Key Switch"
  I:2.0/12  "input from customer Packager Concluded"
  L16:3  TRIG_DELAY_MIN_TIME
  L16:5  CLEARTIME1  "time to clear tracking data"
  L16:6  CLEARTIME5
  L16:7  CLEARTIME6
  L16:8  PASS1PRTLOC
  L16:9  PASS1PROCESSTM
  L16:11  PASS5PROCESSTM
  L16:13  PASS6PROCESSTM
  L23:1  MPCE_ON
  L23:19  TOP_OPT_FAIL_CT
  L23:34  AIR_PRESSURE_FAULT
  L183:2  "simulated part width"
  L187:0  ACQTM1
  L187:1  ACQTM5
  L187:2  ACQTM6
  L187:5  "pass transfer out signals"
  L187:6  "NoErr transfer out signals"
  L187:7  "ins 1 trigger count"
  L190:0  "count of bottom optic width fails"
  L190:1  "count of gap fails"
  L190:2  "I1 blocked triggers"
  L190:4  "count of parts rejected because acquire time ran out"
  L190:5  "count of parts that received a pass signal but previously failed 1"
  L190:6  "count of result signals received with no part present 1"
  L190:7  "count of results received after maximim time reached"
  L190:8  "pass count"
  L190:9  "fail count"
  L190:10  "acquisition count"
  L190:11  "acquisition without result count"
  L190:12  "count of parts results that time out"
  L190:27  "optic alignment pass signal"
  L190:28  "optic alignment fail signal"
  L190:31  "something wrong, can't happen"
  L190:32  "Crazy wrong, can't happen"
  L192:1  BOT_LAST_TIME  "rtc bot belt previous movement event time"
  L192:2  BOT_CYCLE_TIME  "rtc bot belt time between events"
  L192:7  FROM_REAL  "distance from real part signal at optic location"
  L192:8  FROM_TRACKED  "distance from tracked part signal at optic location"
  L192:16  TOP_LAST_TIME  "rtc top belt previous movement event time"
  L192:17  TOP_CYCLE_TIME  "rtc top belt time between events"
  L199:5  ACQTM51
  L199:6  ACQTM52
  L199:7  ACQTM53
  L199:13  DUMP_LONG
  L199:15  ACQTM11
  L199:16  ACQTM12
  L199:17  ACQTM13
  L199:20  RESULTTM1
  L199:22  CLEARTIME5COUNT
  L199:23  CLEARTIME6COUNT
  L199:24  ACQTM61
  L199:25  ACQTM62
  L199:26  ACQTM63
  L199:27  TMSINCETRIG1
  L199:29  TMSINCETRIG5
  L199:30  TMSINCETRIG6
  L199:31  CLEARTIME1COUNT
  L199:32  RESULTTM5
  L199:33  RESULTTM6
  L199:34  MAXACQTM1
  L199:35  MAXACQTM5
  L199:36  MAXACQTM6
  L201:0  CAM_1_MIN_CY
  L201:1  CAM_5_MIN_CY
  L201:2  CAM_6_MIN_CY
  L201:5  "ms since trig 1 is initialized"
  L201:10  "movement from virtual (pos, add)"
  L204:3  "last time between ins 5 triggers"
  L204:7  "last trigger to trigger time"
  L204:13  "This optic signal time"
  L204:14  "Last optic signal time"
  L204:15  "time between optic signals"
  N7:5  "buffer count 6"
  N7:6  "buffer count 1"
  N7:18  PASS5PRTLOC
  N7:19  PASS6PRTLOC
  N10:1  "old ConveyorStatus"
  N10:2  "PowerOn"
  N10:3  "Local Mode On BypassBoxingPLC"
  N10:4  "Boxing Connected Signal"
  N10:5  "BoxJamSignal"
  N10:6  "WaittingOnBoxSig"
  N10:7  "ConveyorFullSig"
  N10:8  "MachineFaultSig"
  N10:9  "Counter Sensor Fault"
  N10:11  "Feeder Track Sensor Blocked"
  N10:12  "Air Pressure Fault"
  N13:0  "Part Inspecting"
  N13:4  "Completed Counter"
  N13:5  "Trigger Position Counter"
  N13:6  "BlowOff Start Counter"
  N13:7  "BlowOff Stop Counter"
  N13:8  "Inspection Command Counter"
  N13:9  "Complete Counter"
  N13:10  "Pass Signal Counter"
  N13:11  "Solenoid Signal Counter"
  N13:12  "Hold Pass Counter"
  N13:13  "Hold Pass Length"
  N16:1  "Bottom Inspection Offset For Tracking"
  N16:3  "Bit Shift Preset"
  N17:5  "Parts In Tube Counter"
  N17:6  "Parts In Tube Limit"
  N17:9  "Bot to Top Transfer Position"
  N17:12  "Trigger to laser Counter"
  N197:1  "maximim acquire time 1"
  N197:5  "Feeder Speed Output Setting"
  N197:10  "pulse distance to keep blow on then turn off feed"
  N197:11  "speed in pps"
  N197:12  "seconds of ontime"
  N197:20/0  "Deformed Head Blowoff Bit to TOP PLC"
  N200:0  RESULTPOS6A
  N200:1  RESULTPOS6B
  N200:2  RESULTPOS5A
  N200:3  RESULTPOS5B
  N200:4  RESULTPOS5C
  N200:5  DUMP_INT
  N200:6  PLATOL  "part location at top optic load"
  N200:7  RESULTPOS5D
  N200:8  RESULTPOS6C
  N200:9  RESULTPOS6D
  N200:10  ACQPOS11
  N200:11  ACQPOS12
  N200:12  ACQPOS13
  N200:14  ACQPOS1  "part acq pos 1"
  N200:15  RESULTPOS1  "result position 1"
  N200:17  RESULTPOS5
  N200:18  RESULTPOS6
  N200:19  ACQPOS5  "part acq pos 5"
  N200:20  ACQPOS6  "part acq pos 6"
  N200:21  ACQPOS51
  N200:22  ACQPOS52
  N200:23  ACQPOS53
  N200:24  ACQPOS61
  N200:25  ACQPOS62
  N200:26  ACQPOS63
  O:0.0/1  "spare"
  O:0.0/5  INS_4_TRIG
  O:0.0/6  "spare"
  O:0.0/11  "Spare"
  O:0.5  "spare"
  O:3.0/0  "Ready-Run signal to Boxer? Always on unless fault?"
  O:3.0/2  "Customers pecies counting done signal (Change Box?)"
  O:3.0/7  "Spare"
  O:3.0/8  "spare"
  PFILE:6  "check for part jams"
  PFILE:10  "Bottom belt HSC"
  PFILE:12  "Top belt HSC"
  Q2:55  END_OF_MAIN
  Q5:94  END_OF_BELTS
  R6:0  "track part location until acquire 1"
  R6:1  "track acquire time 1"
  R6:2  "track part location until acquire 5"
  R6:3  "track acquire time 5"
  R6:5.POS  "Empty Fifo"
  R6:8  "track part location until acquire 6"
  R6:9  "track acquire time 6"
  R21:0  "Trigger Shift Register"
  T20:0  "Trigger On Time"
  U:5  "conveyor"
  U:9  "slow data"
  U:11  "transfered data calcuations from the high speed section"
  U:28  "faults"
  U:29  "speed"
  U:30  "count"
  U:31  "rate calc"
  U:32  "boxer"
  U:33  "bulk pack"
  U:34  "customer boxing unit signals"
  U:35  "cleanup"
  U:95  "HMI interface"

COMMENTS NOT ATTACHED TO A CURRENT RUNG
  F8:13: *************************
    Loads Side Camera Passing data into a bit shift
    *************************
    
    loads passing data bit into passing data bit shift register at the part present cl.
  I:0.0/8: special rung for testing. This rung can simulate a pass signal. It will not be timed correctly.
  B23:0/0: Yet another bit shift load with data in the part position indicating that there was a bottom system part pass as well as a top system part present at this location.
    
    verified works w/bypassed 071910 and unbypassed 072010
  N7:25: 1050
  C5:4: tempory counting to verify pass part count with boxing part count.
  B22:0/0: ***********************
     Bottom Part Syncronizing Logic
    ***********************
    
    This is the point at the bottom of the top conveyor where the part jumps from the bottom conveyor.  This system will then track the part through the top system to the point of the laser optic in order to verify that the part in question has passed the bottom inspection.  I believe that we NEED to include FAILING inspections to eliminate the possibility of a out of position part from passing. LW 072010
  T20:2.ACC: This rung is starting a timer that should be activated directly before the laser optic part presense sensor on the top conveyer and should cause the top optic to be ignored if the bottom camera system didn't pass. however other arrangements must be made if the bottom camera isn't going to be used as is the case with a nut inspection.
  T20:2: The timer used to verify that the part that triggered the top laser optic has passed the bottom camer. needs to be count
  N17:8: ****************************************************************************************************************
    I can not find anywhere in the program where the "Test Spacing From Pickup to Trigger is activated indicating to me that this entire function must not be doing anything in this program at this time.
    ****************************************************************************************************************
  B11:0/0: load part present bit shit with one shot data from the part present sensor
  B3:7/9: ************************************
     The next 3 rungs appear to do nothing
    ***********************************
  B3:6/0: make a bit come on indicating that a part that passed the bottom camera is within  range when crossing the top camera.
  B3:6/1: ***********************
    Part Width and  Location
    ***********************
    
    Calculates the position of parts on the top belt by measureing the part width by calculating the number of belt movement pulses that occure when the optic is blocked and then devides that in half and add that to the optic location in the part presnet bit shift when the top optic is cleared.
  N7:45: not fully functional because of part overlap but measurems the camera responce time when part inspections are not overlaping
  B9:0/[N7:47]: Remove any part present signals outside of expected location
  B9:0/[N7:50]: Remove any part present signals outside of expected location
  F19:0: Counter inside of a high speed counter interrupt counts the number of Bit Shifts that need to be processed in order to move the logic with the parts on the conveyor.
  F8:14: **************
    Bottom Top Camera Trigger
    *************
    
    Trigger Bottom Top Camera
  N10:4: test if boxing is connected
  B3:11/3: After initial delay allow blow two start functioning
  RUNG000150-000011: trigger count
  RUNG000150-000012: wipe stored part data if acq time expires
  RUNG000150-000013: clear data for aquire time expired
  RUNG000150-000014: clear data for time
  RUNG000150-000016: wiped count
  RUNG000150-000018: pass, fail and acquire inputs
  RUNG000150-000025: pass code / Set pass bit in Bit Shift
    captures result position and processing time
    Unlatch pass bit
  RUNG000150-000032: pass count
  RUNG000150-000035: fail count
  RUNG000150-000038: acquire code
  RUNG000150-000039: Grab trigger/acquire position
    Grab acquire time
  RUNG000150-000041: transfer tracked part positon from trigger/acquire to the acquire/result
    capture acquire time
    reset process time
  L14:8: on when ok for run
  L14:3: off when ok to run
  L14:2: off when ok to run
  L14:5: on when ok to run, rear off turns both off
  N7:76: removed relieance on trigger signal
  N197:20/0: Passes deformed head blowoff command to TOP PLC where solenoid output is located.
  N7:47: ***********************************************************************************************************************************************************
    From side
    ***********************************************************************************************************************************************************
    
    removed relieance on trigger signal
  N7:50: ***********************************************************************************************************************************************************
    From top
    ***********************************************************************************************************************************************************
    
    removed relieance on trigger signal
  B3:10/1: prevents momentary signals from box present sensor from tripping the logic for box not present
    
    This is in responce to a problem created by the sensor occasionally turning on as if no box was in its path when there is a box present.
  B3:6/2: IF PROCESSING FAULT OCURES AT COUNTER SENSOR; CLEAR THE BELT OF PASSING DATA
  L14:23: ****************  nEEDS fIXING  **********************
  L14:36: ****************  nEEDS fIXING  **********************
  RUNG000010-000014: ****
                      Zeros out the non passing part count when one passes
    ****
  RUNG000010-000018: Remove any part present signals outside of expected location
  RUNG000125-000014: clear data for time
  RUNG000125-000013: clear data for aquire time expired
  RUNG000125-000012: wipe stored part data if acq time expires
  RUNG000125-000011: trigger count
  RUNG000125-000029: Set pass bit in Bit Shift
    captures result position and processing time
    Unlatch pass bit
  RUNG000125-000027: transfer tracked part positon from trigger/acquire to the acquire/result
    capture acquire time
    reset process time
  RUNG000125-000026: Grab trigger/acquire position
    Grab acquire time
  RUNG000125-000025: pass code / Set pass bit in Bit Shift
    captures result position and processing time
    Unlatch pass bit
  RUNG000125-000018: pass, fail and acquire inputs
  RUNG000125-000016: wiped count
  N7:46: Remove any part present signals outside of expected location

REVISION NOTES
  13: updated count reset
  14: added io moduals
  15: multiple steps toward new hmi integration
  21: test

DATA TABLE (non-zero values as saved)
DATA B3
% B3:0 % 0XA001 0X4000 0X0041 0XA000 0XE10C 0X0362 0X4603 0X0021 0X4007 0X0000
% B3:10 % 0X2041 0X0846 0X2000 0X0000
DATA T4
% .PRE .ACC %
% T4:0 % 300 305
% T4:1 % 150 0
% T4:2 % 32765 0
% T4:3 % 32765 0
% T4:4 % 32765 0
% T4:5 % 180 0
% T4:6 % 10 10
% T4:7 % 150 150
% T4:8 % 150 150
% T4:9 % 50 34
% T4:10 % 200 200
% T4:11 % 150 150
% T4:12 % 44 45
% T4:13 % 6 4
% T4:14 % 180 0
% T4:15 % 150 0
% T4:16 % 11 0
% T4:17 % 100 70
% T4:18 % 120 0
% T4:19 % 300 0
% T4:20 % 200 0
% T4:21 % 200 0
% T4:22 % 200 0
% T4:23 % 50 0
% T4:24 % 50 0
% T4:25 % 50 0
% T4:26 % 250 0
% T4:27 % 250 0
% T4:28 % 250 0
% T4:29 % 5000 0
% T4:30 % 50 50
% T4:31 % 20 0
% T4:32 % 69 0
DATA C5
% .PRE .ACC %
% C5:0 % 32766 0
DATA R6
% .LEN .POS %
% R6:0 % 3 0
% R6:1 % 3 0
% R6:2 % 3 0
% R6:3 % 3 0
% R6:4 % 1250 0
% R6:5 % 1250 0
% R6:6 % 1100 0
% R6:7 % 10 0
% R6:8 % 3 0
% R6:9 % 3 0
% R6:10 % 700 0
% R6:11 % 700 0
% R6:12 % 10 0
% R6:13 % 10 0
% R6:14 % 10 0
% R6:15 % 10 0
% R6:16 % 1100 0
% R6:17 % 700 0
% R6:18 % 700 0
% R6:19 % 10 0
DATA N7
% N7:0 % 1306 3 1022 996 0 0 1 1604 92 75
% N7:10 % 1216 61 1603 1602 1601 1600 3 3 1222 2045
% N7:20 % 1295 3 175 0 0 0 -2 0 0 0
% N7:50 % 1236 0 175 16 0 0 0 1464 12 0
% N7:60 % 1 32767 4012 20 31 0 0 15 30 20
% N7:70 % 0 21 23 27738 32767 0 122 0 16 0
% N7:80 % 0 6 95 0 0 0 5 500 0 0
% N7:90 % 2011 4 4 12 1 0 0 0 0 1600
% N7:100 % 1003 90 110 100 175 25 0 0 0 0
DATA F8
% F8:0 % 18 206.64 23807 499 0.23807
% F8:5 % 4 0 500 1.9 2
% F8:10 % 1 0.08897486 3081 101 63.26563
% F8:15 % 37.73437 4040 2 0 0
% F8:20 % 0 0.02 0 1 0
% F8:25 % 0 932781 0.222 279.6551 848597
% F8:30 % 0 170 0.03 38 852060
% F8:35 % 0 0 0 0 77
% F8:40 % 101 37.73437 0 100 1
% F8:45 % 1 2 0.21455 0 0
% F8:50 % 0 0 1 0 1
% F8:55 % 2000000 -221 0 0 0
% F8:95 % 0 0 0 492 4.92
DATA B9
% B9:130 % 0X0000 0X0000 0X0000 0X0000 0X2000 0X0000 0X0000 0X0000 0X0000 0X8000
% B9:140 % 0X2480 0X0000 0X0000 0X0000 0X0000 0X0000 0X0000 0X0000 0X0000 0X0000
% B9:160 % 0X0000 0X0000 0X0000 0X0000 0X0000 0X0000 0X2000 0X0002 0X0000 0X0000
% B9:170 % 0X0000 0X0000 0X0000 0X2000 0X0000 0X0000 0X0000 0X0000 0X0000 0X0000
% B9:180 % 0X0000 0X0000 0X0000 0X0000 0X0000 0X0002 0X0000 0X0000 0X0000 0X0000
% B9:190 % 0X0010 0X0000 0X0000 0X0000 0X0000 0X0000 0X0000 0X0000 0X0000 0X0000
% B9:200 % 0X2B64 0X2B64 0X0000 0X0010 0X0000 0X2000 0X0000 0X0000 0X0000 0X0000
% B9:220 % 0X0000 0X0000 0X0000 0X0200 0X0000 0X0000 0X0000 0X0000 0X0000 0X0020
% B9:230 % 0X0040 0X0000 0X0000 0X0000 0X0000 0X0000 0X0000 0X0000 0X0000 0X0000
DATA B11
% B11:180 % 0X0000 0X8000 0X0000 0X0000 0X0000 0X0000 0X0000 0X0000 0X0000 0X0000
% B11:240 % 0X0000 0X0000 0X0000 0X4000 0X0000 0X0000 0X0000 0X0000 0X0000 0X0000
DATA B12
% B12:0 % 0X0555 0X0000 0X0000 0X0000 0X0000 0X0000 0X0000 0X0000 0X0000 0X0000
DATA L13
% L13:0 % 308402300 308407124 4824 0 1000
% L13:5 % 2638 47 93 1162124017 1162124017
% L13:10 % 492 79 0 0 0
% L13:15 % -1924744835 -2147483648 2147483647 2147483647 82058
% L13:20 % 514783590 514932830 21377 5 -1924766186
% L13:25 % 514768284 48 250 11 4
% L13:30 % 0 34 0 -1924763091 34
% L13:35 % 1174346533 34 18317 126 1176169897
% L13:40 % 5 0 50 20 0
% L13:45 % 60 600 0 0 15924
% L13:50 % 0 0 0 495000 60
% L13:55 % 42 10 18355 1 50
% L13:60 % 495000 255 48 -1924763139 514919711
% L13:65 % 49 20 1176204078 1176204056 -1924766138
% L13:70 % 1176232488 1176232401 87 2634741 2
% L13:75 % 35391 4 495000 -1924763071 -1924763126
% L13:80 % 55 514919721 150 200 200
% L13:85 % 16 200 50 12531 1000
% L13:90 % 12505 0 0 1000 0
% L13:95 % 60 99000 99000 12542 99000
% L13:100 % 1173535156 1 7 10 8
% L13:105 % 1 1 514768154 5764 514768148
% L13:110 % 6 30 0 514919483 514919479
% L13:115 % 514919487 8 4 514919483 0
% L13:120 % 0 5761 0 30 5761
% L13:125 % 164 19 155494060 137 155494060
% L13:130 % 0 0 -5761 0 0
% L13:135 % 0 1000 111 20 0
% L13:140 % 0 4 20 0 20
% L13:145 % 29761 14877 14881 111 111
% L13:150 % -1538760531 -1538760111 88 0 100
% L13:155 % 420 332 0 0 12985
% L13:160 % 3 2 4 395082 53203921
% L13:165 % 3 189116 95 13 8148
% L13:170 % 55946610 46 44 52 0
% L13:175 % 0 0 10 7 4
% L13:180 % 50841258 25 99000 52866 43242559
% L13:185 % 4324 43242683 4324 43242016 4324
% L13:190 % 4 5 0 0 0
DATA F14
% F14:0 % 710.1306 711.1906 71 71 2064.258
% F14:5 % 26212.8 0 0 0 0
DATA N15
% N15:0 % 6 922 1502 1256 1246 133 100 1169 1018 10
% N15:10 % 63 494 0 0 0 0 1169 0 0 0
DATA L16
% L16:0 % 8 44 11 0 20
% L16:5 % 250 5000 5000 182 19
% L16:10 % 1256 18 2045 6599584 98
% L16:15 % 99 0 0 0 0
DATA B17
% B17:60 % 0XC000 0X0000 0X0000 0X0000 0X0000 0X0000 0X0000 0X0000 0X0000 0X0000
% B17:100 % 0X0000 0X0000 0X0000 0X0000 0X0000 0X0000 0X0000 0X0000 0X1000 0X0000
% B17:110 % 0X4000 0X0000 0X0000 0X0000 0X0000 0X0000 0X0000 0X0000 0X0000 0X0000
% B17:120 % 0X0000 0X0000 0X0000 0X0000 0X0000 0X0000 0X0000 0X2000
DATA B18
% B18:60 % 0XC000 0X0000 0X0000 0X0000 0X0000 0X0000 0X0000 0X0000 0X0000 0X0000
% B18:100 % 0X0000 0X0000 0X0000 0X0000 0X0000 0X0000 0X0000 0X0000 0X0000 0X8240
% B18:110 % 0X0000 0X0400 0X0000 0X0000 0X0000 0X0000 0X0040 0X0000 0X0000 0X0010
% B18:120 % 0X0000 0X0000 0X0000 0X0000 0X0000 0X0000 0X0000 0X2000
DATA L23
% L23:0 % 65535 -65536 -65536 -65536 -65536
% L23:5 % -65536 -65536 2 65535 -65536
% L23:10 % -65536 0 17 10 17
% L23:15 % 0 0 0 0 8
% L23:20 % 0 -65536 -65536 -65536 -65536
% L23:25 % -65536 20 19 20 0
% L23:30 % 0 0 -65536 -65536 -65536
% L23:35 % -65536 -65536 -65536 -65536 -65536
% L23:40 % 16270 18414 0 63266 -65536
% L23:45 % 5062 0 0 0 0
% L23:50 % 0 -65536 -65536 17 -65536
% L23:55 % 33 5079 -65536 0 0
% L23:60 % 0 -65536 -65536 -65536 0
DATA L24
% L24:0 % -65536 122 -65536 222 -65536
% L24:5 % 65535 -65536 -65536 -65536 -65536
% L24:10 % 50 27 0 1 23
% L24:15 % 1198 1030 95 18 30
% L24:20 % 30 -65536 1226 -65536 -65536
% L24:25 % 222 1236 -65536 -65536 222
% L24:30 % 1466 27 10000 -65536 55
% L24:35 % 180 -65536 180 65535 101
% L24:40 % 101 1000 -65536 -65536 10
% L24:45 % 222 192 -65536 0 -65536
% L24:50 % -999 30 10000 65535 900
DATA L42
% L42:0 % 41 0 0 0 0
% L42:5 % 45 45 45 0 0
% L42:20 % 0 0 32766 32766 0
% L42:50 % 0 30
DATA L183
% L183:0 % 1427522383 1427522384 1 1000000000 0
% L183:5 % 59 64 201 0 0
DATA B185
% B185:0 % 0X0200 0X0001 0X0000 0X0000 0X0000 0X0000 0X0000 0X0000 0X0000 0X0000
DATA N186
% N186:0 % 100 0 0 0 0 0 0 0 0 0
DATA L187
% L187:0 % 34 26 497 0 0
% L187:5 % 1063 0 0 0 0
DATA F188
% F188:0 % 6 66 11 44 29
DATA B189
% B189:0 % 0X00F0 0X0000 0X0000 0X0000 0X0000 0X0000 0X0000 0X0000 0X0000 0X0000
DATA L190
% L190:0 % 1 5 0 0 0
% L190:30 % 0 2 0 0 0
DATA B191
% B191:0 % 0X0000 0X0001 0X0000 0X0000 0X0000 0X0000 0X0000 0X0000 0X0000 0X0000
DATA L192
% L192:0 % 1176447793 266932201 5055 269 0
% L192:5 % 100000 36500000 999 999 8
% L192:10 % 0 1 0 78 17
% L192:15 % 1176447720 332250347 860888 268 0
% L192:20 % 180 36500000 0 0 0
DATA F193
% F193:0 % 1.254174 0.315 0.022 6 710
% F193:5 % -0.2825317 0.2 -0.05650635 890.4633 29176.92
% F193:10 % 0.011 0.195 0.165 0.337 710
% F193:15 % -0.2134399 0.25 -0.05335999 582.5885 19089.09
DATA B196
% B196:0 % 0X0C34 0XDFF6 0X0005 0X0000 0X0000 0X0000 0X0000 0X0000 0X0000 0X0000
% B196:30 % 0XE800 0X9BFF 0XEBFF 0XFFDF 0XFFFF 0X0000 0X0000 0X0000 0X0000 0X0000
DATA N197
% N197:0 % 1560 150 500 2500 2500 14417 5555 300 150 0
% N197:10 % 4000 969 4 0 0 0 0 0 0 0
% N197:30 % 15 48 0 0 0 0 0 0 0 0
DATA B198
% B198:0 % 0X0009 0X0000 0X0000 0X0000 0X0000 0X0000 0X0000 0X0000 0X0000 0X0000
DATA L199
% L199:0 % 1 5571998 134 11 3579521
% L199:5 % 0 0 0 5 1049790
% L199:10 % 0 224 10256 556 0
% L199:15 % 0 0 0 278717848 518
% L199:20 % 28295 16430853 5001 5001 0
% L199:25 % 0 0 28329 0 3781224
% L199:30 % 21630086 251 3809367 15030467 111
% L199:35 % 555 555 0 0 0
DATA N200
% N200:0 % 2046 2047 2046 2047 2045 1594 1004 2045 2045 2045
% N200:10 % 0 0 0 1277 178 2046 1000 2045 2045 1218
% N200:20 % 1555 0 0 0 0 0 0 0 0 0
% N200:30 % 0 0 32767 0 0 0 0 0 0 0
DATA L201
% L201:0 % 20 40 40 -3011735 44
% L201:5 % 96629277 0 0 -3010662 0
% L201:10 % 0 0 0 327 43
% L201:15 % 0 43 0 43 36830
DATA B202
% B202:0 % 0X2241 0X0000 0X0001 0X0000 0X0000 0X0000 0X0000 0X0000 0X0000 0X0000
DATA N203
% N203:0 % 115 115 116 333 334 333 444 0 445 444
% N203:10 % 555 556 555 0 0 0 0 0 0 0
DATA L204
% L204:0 % 333 333 333 1362 124
% L204:5 % 2000 2000 462 222 0
% L204:10 % 0 0 0 1327077052 1327077052
% L204:15 % 1327077052 1327077052 1 0 0
% L204:20 % 0 0 33 0 0
% L204:30 % 33 0 0 0 0
DATA F205
% F205:0 % 655.32 655.32 655.32 655.32 0
